Fanuc KAREL source: kb00006.KL

-- PROVISIONAL review KL for V940-1; original PC SHA256 d1ec3fffc12809eba07f74e8151605806068a475769b648d77d8113cf11c29c2
-- Incomplete behavior may be omitted. Consult companion uncertainty JSON. Do not deploy.
PROGRAM KB00006
%NOLOCKGROUP
BEGIN
  -- V9_ZERO_TABLE_METADATA_HINT layout=0002_ascii; no indexed target words; source/name/runtime held
  -- UNRESOLVED_PC offsets 5-12; opcodes 9D,23
  -- UNRESOLVED_PC offsets 17-27; opcodes 9D,22,9D,33,35
  -- UNRESOLVED_PC offsets 32-39; opcodes 9D,23
  -- UNRESOLVED_PC offsets 44-51; opcodes 9D,23
  -- UNRESOLVED_PC offsets 56-90; opcodes 27,22,22,22,22,22,31
  -- UNRESOLVED_PC offsets 95-99; opcodes 7F
END KB00006
